// Mitsubishi GX Works2 project: mitsu_SCADA_PLC_v6   PLC: FX1N/FX1NC

PROGRAM MAIN
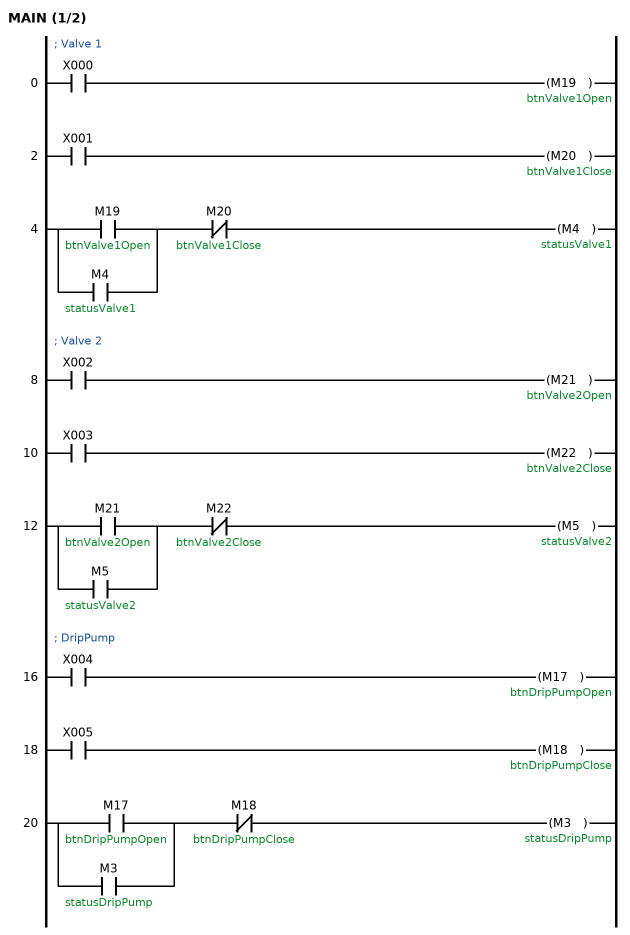
; Valve 1
0     LD      X000
      OUT     M19  ; btnValve1Open
2     LD      X001
      OUT     M20  ; btnValve1Close
4     LD      M19  ; btnValve1Open
      OR      M4  ; statusValve1
      ANI     M20  ; btnValve1Close
      OUT     M4  ; statusValve1
; Valve 2
8     LD      X002
      OUT     M21  ; btnValve2Open
10    LD      X003
      OUT     M22  ; btnValve2Close
12    LD      M21  ; btnValve2Open
      OR      M5  ; statusValve2
      ANI     M22  ; btnValve2Close
      OUT     M5  ; statusValve2
; DripPump
16    LD      X004
      OUT     M17  ; btnDripPumpOpen
18    LD      X005
      OUT     M18  ; btnDripPumpClose
20    LD      M17  ; btnDripPumpOpen
      OR      M3  ; statusDripPump
      ANI     M18  ; btnDripPumpClose
      OUT     M3  ; statusDripPump
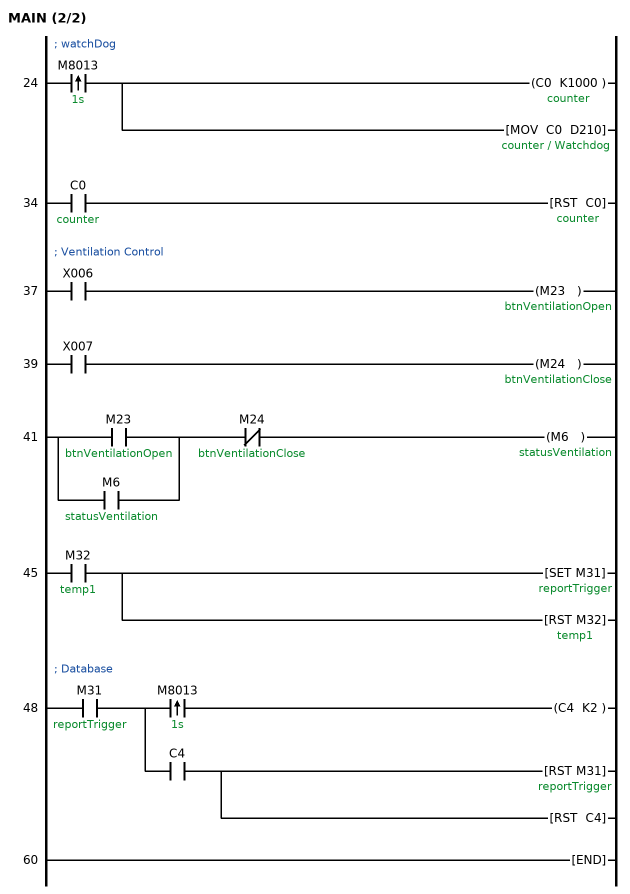
; watchDog
24    LDP     M8013  ; 1s
      OUT     C0 K1000  ; counter
      MOV     C0 D210  ; Watchdog
34    LD      C0  ; counter
      RST     C0  ; counter
; Ventilation Control
37    LD      X006
      OUT     M23  ; btnVentilationOpen
39    LD      X007
      OUT     M24  ; btnVentilationClose
41    LD      M23  ; btnVentilationOpen
      OR      M6  ; statusVentilation
      ANI     M24  ; btnVentilationClose
      OUT     M6  ; statusVentilation
45    LD      M32  ; temp1
      SET     M31  ; reportTrigger
      RST     M32  ; temp1
; Database
48    LD      M31  ; reportTrigger
      MPS
      ANDP    M8013  ; 1s
      OUT     C4 K2
      MPP
      AND     C4
      RST     M31  ; reportTrigger
      RST     C4
60    END
END_PROGRAM

// device comments not shown above
M0  ; statusSystem
M1  ; statusWindow
M2  ; statusDoor
M7  ; statusCoolingFan
M8  ; statusHeater
M9  ; statusLamp
M10  ; btnStart
M11  ; btnStop
M12  ; btnWindowOpen
M13  ; btnWindowClose
M14  ; btnDoorOpen
M15  ; btnDoorClose
M16  ; btnUpdateParameters
M25  ; btnCoolingFanOpen
M26  ; btnCoolingFanClose
M27  ; btnHeaterOpen
M28  ; btnHeaterClose
M29  ; btnLampOpen
M30  ; btnLampClose
D200  ; vFanOpenTime
D201  ; vFanCloseTime
D202  ; cFanOpenTime
D203  ; cFanCloseTime
D204  ; dripIterationTime
D205  ; dripIrrigatedTime
D206  ; setTemperature
D207  ; setMoisture
D208  ; actualTemperature
D209  ; actualMoisture
D211  ; actualTDS
